// TwinCAT 3 PLC project Twee_Pompen
// ProgramVersion: 3.1.4024.0
// libraries:
//   Tc2_Standard, * (Beckhoff Automation GmbH)
//   Tc2_System, * (Beckhoff Automation GmbH)
//   Tc3_Module, * (Beckhoff Automation GmbH)
// project tree:
//   / PlcTask.TcTTO
//   POUs/ MAIN.TcPOU

CONFIGURATION Twee_Pompen
    RESOURCE PLC ON TwinCAT3
        TASK PlcTask(INTERVAL := T#10ms, PRIORITY := 28);
        PROGRAM MAIN WITH PlcTask : MAIN;
    END_RESOURCE
END_CONFIGURATION

// ---- POUs/MAIN.TcPOU
PROGRAM MAIN
VAR
// Inputs
	HoofdSchakelaar AT %I* : BOOL;
    StartDrukknop AT %I* : BOOL;
    StopDrukknop AT %I* : BOOL;
    NiveauSchakelaarLaag AT %I* : BOOL;
    NiveauSchakelaarHoog AT %I* : BOOL;
    Teller: INT := 0;

//Outputs
    Pomp1 AT %Q* : BOOL;
    Pomp2 AT %Q* : BOOL;
	
END_VAR

(*
Twee Pompen (1 regel code + 3regels voor inversie 2 pompen)

Een tank wordt gevuld met twee pompen. 
Om onderhoud te vermijden en de slijtage aan de pompen te spreiden zal men elke pomp om beurten apart laten werken. 
De installatie zal pas werken als een hoofdschakelaar AAN staat.

De pompbeweging wordt gestart ofwel:

    manueel door een startdrukknop
    automatisch door een niveauschakelaar (onderin de tank)

De pompbeweging wordt gestopt ofwel:

    manueel door een stopdrukknop
    automatisch door een niveauschakelaar (bovenaan de tank)
*)

IF HoofdSchakelaar AND (StartDrukknop OR (NOT NiveauSchakelaarHoog AND NiveauSchakelaarLaag)) THEN Teller := (Teller + 1) MOD 2; END_IF;
Pomp1 := (Teller = 0) AND NOT StopDrukknop AND NOT NiveauSchakelaarHoog;
Pomp2 := (Teller = 1) AND NOT StopDrukknop AND NOT NiveauSchakelaarHoog;

END_PROGRAM
